# B&R Automation Studio project testing1
Automation Studio 4.6.3.55 SP; technology packages: mappView 5.6.4

## Configuration Config1

### Task classes (Cpu.sw)
```
Cyclic#4:
  Program <- Program.prg
  Program1 <- Program1.prg
Cyclic#7:
  RevInfo <- RevInfo.RevInfo.prg
Binaries: udbdef, mvLoader, FWRules, TCData, ashwac, arconfig, asfw, ashwd, iomap, User, Role, sysconf
Libraries: fileio, astime, runtime, asieccon, AsBrStr
```

### Hardware
```
X20CP1586 : X20CP1586 v1.5.0.0
  Connector IF2:
    ActivateDevice = 1
    Mode = Manual
    InternetAddress = 192.168.5.16
    SubnetMask = 255.255.255.0
  ConfigurationID = testing1_Config1
  Simulation = 1
  ActivateOpcUa = 1
  OpcUaInformationModels_PV_Version = 1
```

## Logical view

- Visualisation Logical/mappView (not shown)

### Program Logical/Program (IEC)

#### Variables.var
```iecst
VAR
	chicken : USINT;
	time : REAL;
	Speed : INT;
	Temperature : REAL;
END_VAR
```

#### Init.st
```iecst
PROGRAM _INIT
	Speed := 30;
	Temperature := 20;
	chicken := 0;

END_PROGRAM
```

### Program Logical/Program1 (IEC)

#### Variables.var
```iecst
VAR
	nugget : USINT;
END_VAR
```

### RevInfo.var
```iecst
VAR CONSTANT
	revision : STRING[80] := '295e0a3';
	revisionDate : STRING[80] := '2022-05-17 09:26:07 +0800';
	revisionAuthor : STRING[80] := 'Brian Ng';
	branchName : STRING[80] := 'main';
	uncommittedChanges : STRING[80] := ' 35 files changed, 162 insertions(+), 135 deletions(-)';
	buildDate  : STRING[80] := '2022-05-17 09:27:38 +0800';
	buildConfiguration : STRING[80] := 'Config1';
	builder : STRING[80] := 'Brian Ng';
END_VAR
```

- getRevInfo.sh (not shown)

### Program Logical/RevInfo/RevInfo

#### Main.st
```iecst
PROGRAM _INIT

	// Instantiation
	// TODO: Map below into the logger, Machine Settings recipe, or to a diagnostics HMI page
	revision;
	revisionDate;
	revisionAuthor;
	branchName;
	uncommittedChanges;
	buildDate;
	buildConfiguration;
	builder;

END_PROGRAM

PROGRAM _CYCLIC

	// TODO: Tie into to a passive alarm so you won't leave uncommited code in the field.
	UncommittedCodeRunning := (brsstrcmp(ADR(uncommittedChanges),ADR('')) <> 0);

END_PROGRAM

PROGRAM _EXIT

END_PROGRAM
```

### Program Logical/Program2 (IEC)

#### Variables.var
```iecst
VAR
	hello : USINT;
END_VAR
```

#### Init.st
```iecst
PROGRAM _INIT
	hello ;

END_PROGRAM
```

Listed in the project but not available here: Logical/Global.typ, Logical/Global.var, Logical/Libraries
